FUNCTION_BLOCK POU
VAR_INPUT
END_VAR
VAR_OUTPUT
END_VAR
VAR
END_VAR

END_FUNCTION_BLOCK

(* stored: Version 1.1.0.1, ProductVersion 3.1.4022.6
   POU POU: Id {2437f90c-da92-4d9b-94ea-dbb1d6b1d49c}, SpecialFunc None *)
